(* CODESYS project Clock_.xml

Project tree, tasks and I/O mapping:
  program Clock_ [CFC]
*)

// Clock_
PROGRAM Clock_
VAR
	Timezone: TimezoneInformation;
END_VAR

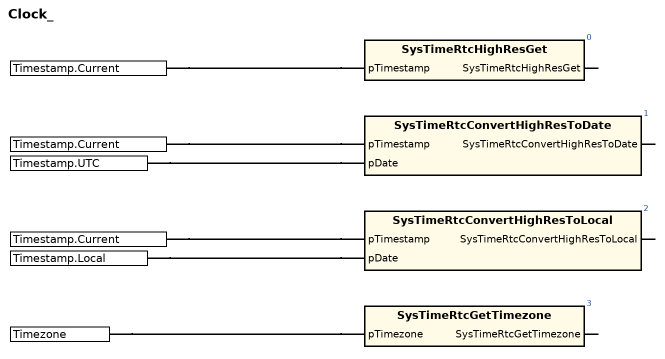
SysTimeRtcHighResGet(pTimestamp := Timestamp.Current);
SysTimeRtcConvertHighResToDate(pTimestamp := Timestamp.Current, pDate := Timestamp.UTC);
SysTimeRtcConvertHighResToLocal(pTimestamp := Timestamp.Current, pDate := Timestamp.Local);
SysTimeRtcGetTimezone(pTimezone := Timezone);

END_PROGRAM
